(* IEC 61131-3 sources: Mizera_Tube/Plc (part 4) *)

(* ---- OUnSu.plc ---- *)
#funcdec "assi.plc"
#funcdec "DynMng.plc"
#funcdec "FBAux.plc"
#funcdec "SupForce.plc"
#funcdec "OSuppFB.plc"

VAR
#include "iof.inc"
#include "usrIof.inc"
#include "cnc.inc"

* Axis support management
* CN7 -> YUVW ( 85,86,87,88 ) Horizontal Supports
* CN8 -> YUVW ( 72,73,74,75 ) Correspoding Vertical Supports

SUP85:        HOR_SUPPORT;
SUP86:        HOR_SUPPORT;
SUP87:        HOR_SUPPORT;
SUP88:        HOR_SUPPORT;

F_TRIG_RES_FOLL:   F_TRIG;
END_VAR

VAR_IN_OUT
#include "usrIol.inc"
#include "mem.inc"
END_VAR

#include "Iol.inc"
#include "usrMem.inc"

FUNCTION HORIZ_SUPP

PATH %cn7

*******************************************************
*     HORIZONTAL FOLLOWIING SUPPORTS MANAGEMENT       *
*******************************************************
CAL  F_TRIG_RES_FOLL (CLK:=PRGRUN_CN0)
LD   F_TRIG_RES_FOLL.Q
OR   Pul_Reset
R    EnWriteBlendSwitch_Hor
R    CmdBlendSwitch_Hor

LDN  PRGRUN_CN0
JMPCN RSTBLEND
     LD   %PLCFLAGS.0
     ST   EnWriteBlendSwitch_Hor
     ST   CmdBlendSwitch_Hor
	 ST   iso_VshapeSecFollow
     ST   Iso_G520HorUnload_Ax85
     ST   Iso_G520HorUnload_Ax86
     ST   Iso_G520HorUnload_Ax87
     ST   Iso_G520HorUnload_Ax88
RSTBLEND:

LD   Reset
OR   EMER_GEN
ST   SUP85.xReset
ST   SUP86.xReset
ST   SUP87.xReset
ST   SUP88.xReset

LD   ISO_SupHor_Init
ST   SUP85.xHoldExem
ST   SUP86.xHoldExem
ST   SUP87.xHoldExem
ST   SUP88.xHoldExem

LDN  OptJogNoAutoHorPrk
ST   SUP85.xEnJogPrk
ST   SUP86.xEnJogPrk
ST   SUP87.xEnJogPrk
ST   SUP88.xEnJogPrk

LD   EnWriteBlendSwitch_Hor
AND  CmdBlendSwitch_Hor
ST   SUP85.xBlendSwitchEn
ST   SUP86.xBlendSwitchEn
ST   SUP87.xBlendSwitchEn
ST   SUP88.xBlendSwitchEn

LD   OptEnabAutoPark
ST   SUP85.xEnabAutoDwn
ST   SUP86.xEnabAutoDwn
ST   SUP87.xEnabAutoDwn
ST   SUP88.xEnabAutoDwn
ST   SUP85.xEnabAutoUp
ST   SUP86.xEnabAutoUp
ST   SUP87.xEnabAutoUp
ST   SUP88.xEnabAutoUp

LD   %ax85.pa22
ST   SUP85.xParkingPos
ST   SUP86.xParkingPos
ST   SUP87.xParkingPos
ST   SUP88.xParkingPos

LD   UnSupHorSafeZone
ST   SUP85.xColiQta
ST   SUP86.xColiQta
ST   SUP87.xColiQta
ST   SUP88.xColiQta

* For Vshape unloading only

LD   iso_VshapeSecFollow
ST   SUP85.xEnSecFollow
ST   SUP86.xEnSecFollow
ST   SUP87.xEnSecFollow
ST   SUP88.xEnSecFollow

LD   VShapeHorOffest
ST   SUP85.xAddFollPos
ST   SUP86.xAddFollPos
ST   SUP87.xAddFollPos
ST   SUP88.xAddFollPos

* [lv, lat, ulv, uhor]=[0,1,2,3]
LD   3
ST   SUP85.xBlendId
ST   SUP86.xBlendId
ST   SUP87.xBlendId
ST   SUP88.xBlendId

LD   iso_G520_Running
ST   SUP85.xEnBldFeed
ST   SUP86.xEnBldFeed
ST   SUP87.xEnBldFeed
ST   SUP88.xEnBldFeed

LD   100
ST   SUP85.xBldFeed
ST   SUP86.xBldFeed
ST   SUP87.xBldFeed
ST   SUP88.xBldFeed

* Horizontal Unloading Speed Control
LD   HorUnloadingFeed
GT   0
AND(
LD   HorUnloadingFeed
LE   100
)
JMPCN _HORFEEDCONTROL
     LD   HorUnloadingFeed
     ST   SUP85.xBldFeed
     ST   SUP86.xBldFeed
     ST   SUP87.xBldFeed
     ST   SUP88.xBldFeed
_HORFEEDCONTROL:

*******************************************************
* Support 1
*******************************************************
LD   %cn7.cc1.2
JMPCN no_support_85

PATH %ax85

LD   Z2Supp_72InParkPos
ST   SUP85.xVerParked

LD   Hold_U_Z2Supp
ST   SUP85.xHoldSuperviAxis

LD   HoldZ2Supp
ST   SUP85.xHoldSuppAxis

LD   SUP72_xParkCmd
ANDN iso_G520_Running
OR   Iso_G520HorUnload_Ax85
AND  %cn0.rc8.0
ST   SUP85.xParkCmd

CAL  SUP85

LD   SUP85.yReqGrant
ANDN ch7_in_ref
ST   usrReqGrantSupHorAx85

LD   SUP85.yHoldMovSupp
ANDN ch7_in_ref
ST   HoldSuppUn_HorAx85

LD   SUP85.yHoldMovSuperv
ANDN ch7_in_ref
ST   Hold_U_SupUnHorAx85

LD   SUP85.yVerForceDwn
ANDN ch7_in_ref
ST   Hor_Ax72_yVerForceDwn

no_support_85:

*******************************************************
* Support 2
*******************************************************
LD   %cn7.cc1.3
JMPCN no_support_86

PATH  %ax86

LD   Z3Supp_73InParkPos
ST   SUP86.xVerParked

LD   Hold_U_Z3Supp
ST   SUP86.xHoldSuperviAxis

LD   HoldZ3Supp
ST   SUP86.xHoldSuppAxis

LD   SUP73_xParkCmd
ANDN iso_G520_Running
OR   Iso_G520HorUnload_Ax86
AND  %cn0.rc8.0
ST   SUP86.xParkCmd

CAL  SUP86

LD   SUP86.yReqGrant
ANDN ch7_in_ref
ST   usrReqGrantSupHorAx86

LD   SUP86.yHoldMovSupp
ANDN ch7_in_ref
ST   HoldSuppUn_HorAx86

LD   SUP86.yHoldMovSuperv
ANDN ch7_in_ref
ST   Hold_U_SupUnHorAx86

LD   SUP86.yVerForceDwn
ANDN ch7_in_ref
ST   Hor_Ax73_yVerForceDwn

no_support_86:

*******************************************************
* Support 3
*******************************************************
LD   %cn7.cc1.4
JMPCN no_support_87

PATH  %ax87

LD   Z4Supp_74InParkPos
ST   SUP87.xVerParked

LD   Hold_U_Z4Supp
ST   SUP87.xHoldSuperviAxis

LD   HoldZ4Supp
ST   SUP87.xHoldSuppAxis

LD   SUP74_xParkCmd
ANDN iso_G520_Running
OR   Iso_G520HorUnload_Ax87
AND  %cn0.rc8.0
ST   SUP87.xParkCmd

CAL  SUP87

LD   SUP87.yReqGrant
ANDN ch7_in_ref
ST   usrReqGrantSupHorAx87

LD   SUP87.yHoldMovSupp
ANDN ch7_in_ref
ST   HoldSuppUn_HorAx87

LD   SUP87.yHoldMovSuperv
ANDN ch7_in_ref
ST   Hold_U_SupUnHorAx87

LD   SUP87.yVerForceDwn
ANDN ch7_in_ref
ST   Hor_Ax74_yVerForceDwn

no_support_87:

*******************************************************
* Support 4
*******************************************************
LD   %cn7.cc1.5
JMPCN no_support_88

PATH  %ax88

LD   Z5Supp_75InParkPos
ST   SUP88.xVerParked

LD   Hold_U_Z5Supp
ST   SUP88.xHoldSuperviAxis

LD   HoldZ5Supp
ST   SUP88.xHoldSuppAxis

LD   SUP75_xParkCmd
ANDN iso_G520_Running
OR   Iso_G520HorUnload_Ax88
AND  %cn0.rc8.0
ST   SUP88.xParkCmd

CAL  SUP88

LD   SUP88.yReqGrant
ANDN ch7_in_ref
ST   usrReqGrantSupHorAx88

LD   SUP88.yHoldMovSupp
ANDN ch7_in_ref
ST   HoldSuppUn_HorAx88

LD   SUP88.yHoldMovSuperv
ANDN ch7_in_ref
ST   Hold_U_SupUnHorAx88

LD   SUP88.yVerForceDwn
ANDN ch7_in_ref
ST   Hor_Ax75_yVerForceDwn

no_support_88:

END_FUNCTION

(* ---- pageplc.plc ---- *)
#include "iol.inc"

VAR
appoggio:        BOOL;
TP_Tab_Note:     TP;
END_VAR

*/ pop out page to select mode after reset */

FUNCTION PAGE_PLC

LD     HMI_PagePop
ANDN   %PLCFLAGS.8
ANDN(
    LD     %Uipl.Page
    EQ     171501
)
JMPCN  POP_WIND_STATE
    LD     171501
    ST     %PlcPage

    LD     1
    S      %ChangePlcPageFlags.3

    LD     1400
    ST     %WidthUiplDlg

    LD     400
    ST     %HeightUiplDlg

    LD     1
    ST     %ChangePlcPage
JMPC   COM_WIND_STATE
POP_WIND_STATE:
    LD     0
    ST     %ChangePlcPage
COM_WIND_STATE:

LD HMI_Ret2Loader
ANDN(
    LD     %Uipl.Page
    EQ     171502           ** Ret2Load.str
)
JMPCN  Skip_Ret2Load
    LD     171502
    ST     %PlcPage

    LD     1
    S      %ChangePlcPageFlags.3

    LD     1400
    ST     %WidthUiplDlg

    LD     400
    ST     %HeightUiplDlg

    LD     1
    ST     %ChangePlcPage
JMPC   COM_WIND_STATE2
Skip_Ret2Load:
    LD     0
    ST     %ChangePlcPage
COM_WIND_STATE2:

LDN    %cn0.rc8.0
JMPCN  PGMNORUNNING
    LD     %PLCFLAGS.0
    ST     Gui_btn_NoGear
    ST     Gui_btn_Gear
    ST     HMI_PagePop
    ST     HMI_Ret2Loader
PGMNORUNNING:

LD     %Uipl.Page
EQ     171501
JMPCN  CLRPAGEREQ
    LD     %PLCFLAGS.0
    ST     HMI_PagePop
CLRPAGEREQ:

LD     %Uipl.Page
EQ     171502
JMPCN  CLRPAGEREQ2
    LD     %PLCFLAGS.0
    ST     HMI_Ret2Loader
CLRPAGEREQ2:

END_FUNCTION

(* ---- Pneumat.plc ---- *)
*******************************************************************************
*   PNEUMAT.PLC
*   ESAutomotion
*   LASER machine
*******************************************************************************
VAR
#include "Cnc.inc"

appoggio:                       BOOL;       * Appoggio
TON_NOARIA:                     TON;        * Manca aria compressa
Strobe_Funz_M493:               BOOL;
Strobe_Funz_M494:               BOOL;
Memo_Aria_ass_taglio_da_Funz_M: BOOL;       * Memoria Aria assistenza al taglio da Funzione M
Aria_ass_taglio_in_Piercing:    BOOL;       * Aria assistenza al taglio in Piercing
R_TRIG493:                      R_TRIG;     * Fronte di salita M493 Attivazione Aria assistenza al taglio
R_TRIG494:                      R_TRIG;     * Fronte di salita M494 Disattivazione Aria assistenza al taglio
Test_Aria_ass_taglio_da_GUI     AT  %LsGui18.1;     *Test Aria assistenza al taglio da GUI
Test_Aria_ugello_da_GUI         AT  %LsGui18.2;     * Test Aria ugello da GUI
END_VAR

#include "Iol.inc"

VAR_IN_OUT
#include "mem.inc"
END_VAR

*******************************************************************************
*   Gestione Impianto Pneumatico
*******************************************************************************
FUNCTION Pneumatico

*******************************************************************************
* Allarme: bassa pressione aria impianto
*******************************************************************************
LDN  I_I_PRESSIONE_ARIA_IMPIANTO   ** Pressione aria Impianto OK
ST   appoggio                      ** Appoggio

CAL  TON_NOARIA(IN=appoggio, PT=1000) ** Manca aria compressa

LD   TON_NOARIA.Q
S    %PLCerr6.1

LD   RESET_ALLARMI                 ** M100.4  Cancellazione allarmi attiva
R    %PLCerr6.1                            ** PLC Err 193 Bassa pressione aria impianto

*******************************************************************************
* Allarme: bassa pressione aria banco
*******************************************************************************
LDN  I_I_PRESSIONE_ARIA_BANCO      ** Pressione aria Banco OK
S    %PLCerr6.2                            ** PLC Err 194 Bassa pressione aria banco

LD   RESET_ALLARMI                 ** M100.4  Cancellazione allarmi attiva
R    %PLCerr6.2                            ** PLC Err 194 Bassa pressione aria banco

*******************************************************************************
* Aria ugello : M498\M497 : Dis\Attivazione (IN Gas.plc)
*******************************************************************************
LD   GAS_prun                      ** M107.1 Cutting gas active from part program
ANDN %PlcOp0.2                     ** DryRun
ANDN PRGSTOP_CN0                   ** (cn0.rc8.1)  Programma interrotto CN0
OR   Test_Aria_ugello_da_GUI       ** Test Aria ugello da GUI
ST   O_O_EV_ARIA_UGELLO            ** Elettrovalvola aria ugello

*******************************************************************************
* Aria assistenza al taglio : M494\M493 : Dis\Attivazione
*******************************************************************************
LD   %cn0.rc9                               ** Channel 0 M-Functions register
EQ   493
AND  %cn0.rc8.4                             ** Channel 0 M-Functions Strobe
ST   Strobe_Funz_M493

CAL R_TRIG493(CLK=Strobe_Funz_M493) ** Fronte di salita M493 Attivazione Aria assistenza al taglio

LD   %cn0.rc9                               ** Channel 0 M-Functions register
EQ   494
AND  %cn0.rc8.4                             ** Channel 0 M-Functions Strobe
ST   Strobe_Funz_M494

CAL  R_TRIG494(CLK=Strobe_Funz_M494) ** Fronte di salita M494 Disattivazione Aria assistenza al taglio

LD   R_TRIG493.Q
S    Memo_Aria_ass_taglio_da_Funz_M ** Memoria Aria assistenza al taglio da Funzione M
LD   R_TRIG494.Q
ORN  MACCHINA_OK                   ** M100.1  Macchina OK
OR   RESET_MACCHINA                ** M100.2  Reset macchina
R    Memo_Aria_ass_taglio_da_Funz_M ** Memoria Aria assistenza al taglio da Funzione M

LD   %TabLsr0.L_UserInt1
EQ   0
ST   Aria_ass_taglio_in_Piercing   ** Aria assistenza al taglio in Piercing

LD   Memo_Aria_ass_taglio_da_Funz_M ** Memoria Aria assistenza al taglio da Funzione M
OR   Aria_ass_taglio_in_Piercing   ** Aria assistenza al taglio in Piercing
AND(
LD   PRGRUN_CN0                    ** M0.0 cn0.rc8.0  Programma in corso
ANDN %PlcOp0.2                     ** DryRun
ANDN PRGSTOP_CN0                   ** (cn0.rc8.1)  Programma interrotto CN0
ANDN ExeAuxMode                    ** (gPlc0.29)Esecuzione ausiliaria 1000.PGM
)
OR   Test_Aria_ass_taglio_da_GUI   ** Test Aria assistenza al taglio da GUI
ST   O_O_EV_ASSISTENZA_TAGLIO      ** Elettrovalvola assistenza taglio

*******************************************************************************
*Segnalazioni per Aggiornamento pagina video
*******************************************************************************
LD   O_O_EV_ARIA_UGELLO            ** Elettrovalvola aria ugello
ST   GasYV23LED                    ** (LsPlc11.12) LED nozzle air

LD   O_O_EV_ASSISTENZA_TAGLIO      ** Elettrovalvola assistenza taglio
ST   GasYV24LED                    ** (LsPlc11.13) LED cut air assistance

END_FUNCTION

(* ---- remcon.plc ---- *)
#include "Iol.inc"

VAR
#include "Cnc.inc"
#include "RemContr.inc"
END_VAR

VAR
DryrunSig                  AT %PlcOp0.2 ; ** DryRun
HoldingZ                   AT %ax29.ra0.1;                  * %ax29.ra0.1 holding Z axis
HoldingX                   AT %ax27.ra0.1;                  * %ax27.ra0.1 holding X axis
HoldingY                   AT %ax28.ra0.1;                  * %ax29.ra0.1 holding Y axis
END_VAR

FUNCTION REMOTE_DISPLAY
******************************************************************************
* THE AXIS DISPLAY
******************************************************************************
LD   %ax30.ra4                   *U position Yang
DIV  10
ST   X_AXIS_POSITION

LD   %ax28.ra4
DIV  10
ST   Y_AXIS_POSITION

LD   %ax29.ra4
DIV  10
ST   Z_AXIS_POSITION

LD      HoldingZ                   ** %ax29.ra0.1 holding Z axis
JMPCN   Z_HOLDING
LD      4
ST      LineZaxis                  ** XhcApp.Xhc_LineIdx3 Feedrate and mode
JMP     END_AZ
Z_HOLDING:
LD      1
ST      LineZaxis                  ** XhcApp.Xhc_LineIdx3 Feedrate and mode
END_AZ:

LD      HoldingX                   ** %ax27.ra0.1 holding X axis
JMPCN   X_HOLDING
LD      5
ST      LineXaxis                  ** XhcApp.Xhc_LineIdx1 X axis quote
JMP     END_AX
X_HOLDING:
LD      2
ST      LineXaxis                  ** XhcApp.Xhc_LineIdx1 X axis quote
END_AX:

LD      HoldingY                   ** %ax29.ra0.1 holding Y axis
JMPCN   Y_HOLDING
LD      6
ST      LineYaxis                  ** XhcApp.Xhc_LineIdx2 Y axis quote
JMP     END_AY
Y_HOLDING:
LD      3
ST      LineYaxis                  ** XhcApp.Xhc_LineIdx2 Y axis quote
END_AY:

******************************************************************************
* THE FEEDRATE DISPLAY
******************************************************************************
LD       DryrunSig                 ** %PlcOp0.2 Dry signal
AND      BCI_TAR                   * rc0.8  Selettore modi operativi su REF (taratura)
JMPCN    DRY_REF
LD       12
ST       LineFeed                  ** XhcApp.Xhc_LineIdx0 Z axis quote
JMP      END_CONDITION
DRY_REF:

LDN      DryrunSig                 ** %PlcOp0.2 Dry signal
AND      BCI_TAR                   * rc0.8  Selettore modi operativi su REF (taratura)
JMPCN    NOTDRY_REF
LD       7
ST       LineFeed                  ** XhcApp.Xhc_LineIdx0 Z axis quote
JMP      END_CONDITION
NOTDRY_REF:

LD       DryrunSig                 ** %PlcOp0.2 Dry signal
AND      BCI_MAN                   * rc0.9  Selettore modi operativi su JOG (manuale)
JMPCN    DRY_JOG
LD       13
ST       LineFeed                  ** XhcApp.Xhc_LineIdx0 Z axis quote
JMP      END_CONDITION
DRY_JOG:

LDN      DryrunSig                 ** %PlcOp0.2 Dry signal
AND      BCI_MAN                   * rc0.9  Selettore modi operativi su JOG (manuale)
JMPCN    NOTDRY_JOG
LD       8
ST       LineFeed                  ** XhcApp.Xhc_LineIdx0 Z axis quote
JMP      END_CONDITION
NOTDRY_JOG:

LD       DryrunSig                 ** %PlcOp0.2 Dry signal
AND      BCI_INC                   * rc0.10  Selettore modi operativi su INC (inc.fissi)
JMPCN    DRY_INC
LD       14
ST       LineFeed                  ** XhcApp.Xhc_LineIdx0 Z axis quote
JMP      END_CONDITION
DRY_INC:

LDN      DryrunSig                 ** %PlcOp0.2 Dry signal
AND      BCI_INC                   * rc0.10  Selettore modi operativi su INC (inc.fissi)
JMPCN    NOTDRY_INC
LD       9
ST       LineFeed                  ** XhcApp.Xhc_LineIdx0 Z axis quote
JMP      END_CONDITION
NOTDRY_INC:

LD       DryrunSig                 ** %PlcOp0.2 Dry signal
AND      BCI_MDI                   * rc0.11  Selettore modi operativi su MDI (semiautom)
JMPCN    DRY_MDI
LD       15
ST       LineFeed                  ** XhcApp.Xhc_LineIdx0 Z axis quote
JMP      END_CONDITION
DRY_MDI:

LDN      DryrunSig                 ** %PlcOp0.2 Dry signal
AND      BCI_MDI                   * rc0.11  Selettore modi operativi su MDI (semiautom)
JMPCN    NOTDRY_MDI
LD       10
ST       LineFeed                  ** XhcApp.Xhc_LineIdx0 Z axis quote
JMP      END_CONDITION
NOTDRY_MDI:

LD       DryrunSig                 ** %PlcOp0.2 Dry signal
AND      BCI_AUT                   * rc0.12  Selettore modi operativi su AUT (automatic)
JMPCN    DRY_AUT
LD       16
ST       LineFeed                  ** XhcApp.Xhc_LineIdx0 Z axis quote
JMP      END_CONDITION
DRY_AUT:

LDN      DryrunSig                 ** %PlcOp0.2 Dry signal
AND      BCI_AUT                   * rc0.12  Selettore modi operativi su AUT (automatic)
JMPCN    NOTDRY_AUT
LD       11
ST       LineFeed                  ** XhcApp.Xhc_LineIdx0 Z axis quote

NOTDRY_AUT:

END_CONDITION:

END_FUNCTION

(* ---- RemContr.plc ---- *)
*******************************************************************************
*   RemContR.plc
*   ESAutomotion
*   LASER machine
*   Remote Controller Manag
*******************************************************************************
#funcdec "FLP.plc"

VAR
#include "RemContr.inc"
END_VAR

#include "Iol.inc"

VAR_IN_OUT
#include "mem.inc"
END_VAR

FUNCTION   REMOTE_CONTROLLER

(* ---- resmach.plc ---- *)
*******************************************************************************
*   RESMACH.PLC
*   ESAutomotion
*   LASER machine
*******************************************************************************
*
* Reset function
* There is update:
* To Reset Axes with TON maybe OK, but CN Reset should check real feedback
* Res_Ch3 is also used to xReset CN4 on this machine
*
* Reset must be:
* 1) Disable gearing to unlock real axes from virtual axes,
* 2) Reset channel 3 4
* 3) Reset channel 0 2 5
*******************************************************************************
#funcdec "assi.plc"
#funcdec "cnc.plc"

VAR
#include "assi.inc"
#include "cnc.inc"

END_VAR

VAR_IN_OUT
#include "mem.inc"
END_VAR

#include "iol.inc"

VAR
RTRIG_RESET:        R_TRIG;
TON_RES_AXES:       TON;
TON_RESCH3:         TON;
TON_RESCH0:         TON;
ResetCh0Ok:         BOOL;
ResetCh3Ok:         BOOL;
check_ch3:          BOOL;
END_VAR

*******************************************************************************
FUNCTION  MACHINE_RESET

LDN  %cn0.rc8.0
ANDN %cn0.rc8.1
ST   ResetCh0Ok

LDN  %cn3.rc8.0
ANDN %cn3.rc8.1
ST   ResetCh3Ok

CAL  RTRIG_RESET(CLK:=ResetMach)          * Reset pushbutton

LD   RTRIG_RESET.Q
S    Res_Axes

CAL  TON_RES_AXES(IN:=Res_Axes,PT:=200)
LD   TON_RES_AXES.Q
***OR(
***LD   ResetCh0Ok
***ANDN ResetCh3Ok
***)
R    Res_Axes
R    check_ch3
S    Res_Ch3

* In Main, not to allow START with any Res_

CAL  TON_RESCH3(IN:=Res_Ch3,PT:=200)
LD   TON_RESCH3.Q
S    check_ch3
R    Res_Ch3

LD   check_ch3
AND  %cn3.rc8.21
R    check_ch3
S    Res_Ch0

CAL  TON_RESCH0(IN:=Res_Ch0,PT:=200)
LD   TON_RESCH0.Q
R    Res_Ch0

END_FUNCTION

(* ---- SupLdCy.plc ---- *)
#funcdec "FBSuppor.plc"
#funcdec "assi.plc"
#funcdec "DynMng.plc"
#funcdec "FBAux.plc"
#funcdec "SupForce.plc"
#funcdec "suppFB.plc"

#include "Iol.inc"
#include "usrMem.inc"

VAR
#include "iof.inc"
#include "usrIof.inc"
#include "cnc.inc"

SUPPORT_1:     TUBE_SUPPORT;
SUPPORT_2:     TUBE_SUPPORT;
SUPPORT_3:     TUBE_SUPPORT;
SUPPORT_4:     TUBE_SUPPORT;
SUPPORT_5:     TUBE_SUPPORT;
SUPPORT_6:     TUBE_SUPPORT;
SUPPORT_7:     TUBE_SUPPORT;
END_VAR

VAR_IN_OUT
#include "usrIol.inc"
#include "mem.inc"
END_VAR

FUNCTION LOAD_CYLINDER_SUPPORTS

*******************************************************
*           CYLINDER SUPPORTS MANAGEMENT              *
*******************************************************
LD   SUPPORTS_JogPlus
ST   SUPPORTS_JogPlusLed

LD   SUPPORTS_JogMinus
ST   SUPPORTS_JogMinusLed

LD   ALWAYS_ONE
ST   SUPPORT_1.xUaxDir
ST   SUPPORT_2.xUaxDir
ST   SUPPORT_3.xUaxDir
ST   SUPPORT_4.xUaxDir

LD   PosUMis
ST   SUPPORT_1.xPosU
ST   SUPPORT_2.xPosU
ST   SUPPORT_3.xPosU
ST   SUPPORT_4.xPosU

LD   ThreshLoadingSupDown
ST   SUPPORT_1.xSuperviseOft
ST   SUPPORT_2.xSuperviseOft
ST   SUPPORT_3.xSuperviseOft
ST   SUPPORT_4.xSuperviseOft

LDN  I_I_EMERGENZA                ** Machine OK (no EMERG.)
ST   SUPPORT_1.xEmerg
ST   SUPPORT_2.xEmerg
ST   SUPPORT_3.xEmerg
ST   SUPPORT_4.xEmerg

LD   ch0_in_aut                   ** channel 0 in aut
ST   SUPPORT_1.xAuto
ST   SUPPORT_2.xAuto
ST   SUPPORT_3.xAuto
ST   SUPPORT_4.xAuto

LD   I_I_PRESSIONE_ARIA_IMPIANTO
ST   SUPPORT_1.xAirPressure
ST   SUPPORT_2.xAirPressure
ST   SUPPORT_3.xAirPressure
ST   SUPPORT_4.xAirPressure

LD   Reset                        ** Reset Command
OR   Start_Ch0                    ** Start Request to Ch0
ST   SUPPORT_1.xReset
ST   SUPPORT_2.xReset
ST   SUPPORT_3.xReset
ST   SUPPORT_4.xReset

LD   TimeOutPistonDown
ST   SUPPORT_1.xTimeOut
ST   SUPPORT_2.xTimeOut
ST   SUPPORT_3.xTimeOut
ST   SUPPORT_4.xTimeOut

*******************************************************
*                      SUPPORT 1                      *
*******************************************************
LD   I_I_Support_1_Dwn            ** M50.7 Support 1 Down Sensor
ST   SUPPORT_1.xSensorDwn

LD   I_I_Support_1_Up
ST   SUPPORT_1.xSensorOpen

LD   SUPPORTS_S1_Selected
AND  SUPPORTS_JogPlus
ST   SUPPORT_1.xManualUp

LD   SUPPORTS_S1_Selected
AND  SUPPORTS_JogMinus
ST   SUPPORT_1.xManualDwn

LD   Fun_M724_Ch0                 ** Auto Up command for supports
OR   Fun_M733_Ch0
ANDN yActivatedCyCom_51
ST   SUPPORT_1.xAutoUp

LD   Fun_M725_Ch0                 ** Auto Up command for supports
OR   yActivatedCyCom_51
ST   SUPPORT_1.xAutoDwn

LD   SUPPORT_1_AutoEnable
ST   SUPPORT_1.xEnable

LD   SUPPORT_1_Quota
ST   SUPPORT_1.xLimitQuota

CAL  SUPPORT_1

LD   SUPPORT_1.yEvUp
ST   O_O_Ev_Support1_Up

LD   SUPPORT_1.yEvDwn
ST   O_O_Ev_Support1_Dwn

LD   SUPPORT_1.yAlarmDwn
ST   SUPPORT_1_AlarmDwn
ST   %PLCerr21.0

*******************************************************
*                      SUPPORT 2                      *
*******************************************************
LD   I_I_Support_2_Dwn             ** M50.8 Support 2 Down Sensor
ST   SUPPORT_2.xSensorDwn

LD   I_I_Support_2_Up              ** PLCFLAGS.1  Flag sempre stato on
ST   SUPPORT_2.xSensorOpen

LD   SUPPORTS_S2_Selected
AND  SUPPORTS_JogPlus
ST   SUPPORT_2.xManualUp

LD   SUPPORTS_S2_Selected
AND  SUPPORTS_JogMinus
ST   SUPPORT_2.xManualDwn

LD   Fun_M724_Ch0                  ** Auto Up command for supports
OR   Fun_M734_Ch0
ANDN yActivatedCyCom_52
ST   SUPPORT_2.xAutoUp

LD   Fun_M725_Ch0                  ** Auto Up command for supports
OR   yActivatedCyCom_52
ST   SUPPORT_2.xAutoDwn

LD   SUPPORT_2_AutoEnable
ST   SUPPORT_2.xEnable

LD   SUPPORT_2_Quota
ST   SUPPORT_2.xLimitQuota

CAL  SUPPORT_2

LD   SUPPORT_2.yAlarmDwn
ST   SUPPORT_2_AlarmDwn
ST   %PLCerr21.1

LD   SUPPORT_2.yEvUp
ST   O_O_Ev_Support2_Up

LD   SUPPORT_2.yEvDwn
ST   O_O_Ev_Support2_Dwn

*******************************************************
*                      SUPPORT 3                      *
*******************************************************
LD   I_I_Support_3_Dwn             ** M50.9 Support 3 Down Sensor
ST   SUPPORT_3.xSensorDwn

LD   I_I_Support_3_Up
ST   SUPPORT_3.xSensorOpen

LD   SUPPORTS_S3_Selected
AND  SUPPORTS_JogPlus
ST   SUPPORT_3.xManualUp

LD   SUPPORTS_S3_Selected
AND  SUPPORTS_JogMinus
ST   SUPPORT_3.xManualDwn

LD   Fun_M724_Ch0                  ** Auto Up command for supports
OR   Fun_M735_Ch0
ANDN yActivatedCyCom_53
ST   SUPPORT_3.xAutoUp

LD   Fun_M725_Ch0                  ** Auto Up command for supports
OR   yActivatedCyCom_53
ST   SUPPORT_3.xAutoDwn

LD   SUPPORT_3_AutoEnable
ST   SUPPORT_3.xEnable

LD   SUPPORT_3_Quota
ST   SUPPORT_3.xLimitQuota

CAL  SUPPORT_3

LD   SUPPORT_3.yAlarmDwn
ST   SUPPORT_3_AlarmDwn
ST   %PLCerr21.2

LD   SUPPORT_3.yEvUp
ST   O_O_Ev_Support3_Up

LD   SUPPORT_3.yEvDwn
ST   O_O_Ev_Support3_Dwn

*******************************************************
*                      SUPPORT 4                      *
*******************************************************
LD   I_I_Support_4_Dwn             ** M50.10 Support 4 Down Sensor
ST   SUPPORT_4.xSensorDwn

LD   I_I_Support_4_Up              ** PLCFLAGS.1  Flag sempre stato on
ST   SUPPORT_4.xSensorOpen

LD   SUPPORTS_S4_Selected
AND  SUPPORTS_JogPlus
ST   SUPPORT_4.xManualUp

LD   SUPPORTS_S4_Selected
AND  SUPPORTS_JogMinus
ST   SUPPORT_4.xManualDwn

LD   Fun_M724_Ch0                  ** Auto Up command for supports
OR   Fun_M736_Ch0
ANDN yActivatedCyCom_54
ST   SUPPORT_4.xAutoUp

LD   Fun_M725_Ch0                  ** Auto Up command for supports
OR   yActivatedCyCom_54
ST   SUPPORT_4.xAutoDwn

LD   SUPPORT_4_AutoEnable
ST   SUPPORT_4.xEnable

LD   SUPPORT_4_Quota
ST   SUPPORT_4.xLimitQuota

CAL  SUPPORT_4

LD   SUPPORT_4.yAlarmDwn
ST   SUPPORT_4_AlarmDwn
ST   %PLCerr21.3

LD   SUPPORT_4.yEvUp
ST   O_O_Ev_Support4_Up

LD   SUPPORT_4.yEvDwn
ST   O_O_Ev_Support4_Dwn

*******************************************************
*                    HOLD CONDITION                   *
*******************************************************
LD   %PLCerr21.0
OR   %PLCerr21.1
OR   %PLCerr21.2
OR   %PLCerr21.3
OR   %PLCerr21.4
OR   %PLCerr21.5
OR   %PLCerr21.6
OR   SUPPORT_1.yHoldMovSuperv
OR   SUPPORT_2.yHoldMovSuperv
OR   SUPPORT_3.yHoldMovSuperv
OR   SUPPORT_4.yHoldMovSuperv
ST   M_HoldAx_U

LD   I_I_Support_1_Dwn
AND  I_I_Support_2_Dwn
AND  I_I_Support_3_Dwn
AND  I_I_Support_4_Dwn
*AND  I_I_Support_5_Dwn
*AND  I_I_Support_6_Dwn
*AND  I_I_Support_7_Dwn
ST   All_Sup_DWN

END_FUNCTION

(* ---- SuUnCy.plc ---- *)
*******************************************************
*  Motor-cylinder Composite Support (Cylinder Part)   *
*  Supports Up/Dwn Conditions Based On Motor Part     *
*******************************************************
#funcdec "FBSuppor.plc"
#funcdec "assi.plc"
#funcdec "DynMng.plc"
#funcdec "FBAux.plc"
#funcdec "SupForce.plc"
#funcdec "suppFB.plc"

#include "Iol.inc"
#include "usrMem.inc"

VAR
#include "iof.inc"
#include "usrIof.inc"
#include "cnc.inc"

SUPPORT_71:     TUBE_SUPPORT;
SUPPORT_72:     TUBE_SUPPORT;
SUPPORT_73:     TUBE_SUPPORT;
SUPPORT_74:     TUBE_SUPPORT;
SUPPORT_75:     TUBE_SUPPORT;
END_VAR

VAR_IN_OUT
#include "usrIol.inc"
#include "mem.inc"
END_VAR

FUNCTION UN_CYLINDER_SUPPORTS
*******************************************************
*    UNLOAD CYLINDER SUPPORTS MANAGEMENT              *
*******************************************************
LD   UNSUPPORTS_JogPlus
ST   UNSUPPORTS_JogPlusLed

LD   UNSUPPORTS_JogMinus
ST   UNSUPPORTS_JogMinusLed

LD   SupervisePos_X1
ST   SUPPORT_71.xPosU
ST   SUPPORT_72.xPosU
ST   SUPPORT_73.xPosU
ST   SUPPORT_74.xPosU
ST   SUPPORT_75.xPosU

LDN  I_I_EMERGENZA
ST   SUPPORT_71.xEmerg
ST   SUPPORT_72.xEmerg
ST   SUPPORT_73.xEmerg
ST   SUPPORT_74.xEmerg
ST   SUPPORT_75.xEmerg

LD   ch0_in_aut
ST   SUPPORT_71.xAuto
ST   SUPPORT_72.xAuto
ST   SUPPORT_73.xAuto
ST   SUPPORT_74.xAuto
ST   SUPPORT_75.xAuto

LD   I_I_PRESSIONE_ARIA_IMPIANTO
ST   SUPPORT_71.xAirPressure
ST   SUPPORT_72.xAirPressure
ST   SUPPORT_73.xAirPressure
ST   SUPPORT_74.xAirPressure
ST   SUPPORT_75.xAirPressure

LD   Reset
OR   Start_Ch0
ST   SUPPORT_71.xReset
ST   SUPPORT_72.xReset
ST   SUPPORT_73.xReset
ST   SUPPORT_74.xReset
ST   SUPPORT_75.xReset

LD   TimeOutPistonDown
ST   SUPPORT_71.xTimeOut
ST   SUPPORT_72.xTimeOut
ST   SUPPORT_73.xTimeOut
ST   SUPPORT_74.xTimeOut
ST   SUPPORT_75.xTimeOut

*******************************************************
* Support On Ax71
*******************************************************
LD   I_I_SUPPORT_71_Dwn
ST   SUPPORT_71.xSensorDwn

LD   I_I_SUPPORT_71_Up
ST   SUPPORT_71.xSensorOpen

LD   SUPPORTS_S71_Selected
AND  UNSUPPORTS_JogPlus
ST   SUPPORT_71.xManualUp

LD   SUPPORTS_S71_Selected
AND  UNSUPPORTS_JogMinus
ST   SUPPORT_71.xManualDwn

LDN  Hold_U_Z1Supp
ANDN SUP71_xParkCmd
ANDN yActivatedCyCom_71
ST   SUPPORT_71.xAutoUp

LD   Hold_U_Z1Supp
OR   SUP71_xParkCmd
OR   yActivatedCyCom_71
ST   SUPPORT_71.xAutoDwn

LD   SUPPORT_71_AutoEnable
ST   SUPPORT_71.xEnable

LD   OffsetUnSuppDwn_71
ST   SUPPORT_71.xSuperviseOft

LD   U_Posit_Z1_Down
ST   SUPPORT_71.xLimitQuota

CAL  SUPPORT_71

LD   SUPPORT_71.yEvUp
ST   O_O_Ev_Support71_Up

LD   SUPPORT_71.yEvDwn
ST   O_O_Ev_Support71_Dwn

LD   SUPPORT_71.yAlarmDwn
ST   %PLCerr20.4

*******************************************************
* Support On Ax72
*******************************************************
LD   I_I_SUPPORT_72_Dwn
ST   SUPPORT_72.xSensorDwn

LD   I_I_SUPPORT_72_Up
ST   SUPPORT_72.xSensorOpen

LD   SUPPORTS_S72_Selected
AND  UNSUPPORTS_JogPlus
ST   SUPPORT_72.xManualUp

LD   SUPPORTS_S72_Selected
AND  UNSUPPORTS_JogMinus
ST   SUPPORT_72.xManualDwn

LDN  Hold_U_Z2Supp
ANDN SUP72_xParkCmd
ANDN yActivatedCyCom_72
ST   SUPPORT_72.xAutoUp

LD   Hold_U_Z2Supp
OR   SUP72_xParkCmd
OR   yActivatedCyCom_72
ST   SUPPORT_72.xAutoDwn

LD   SUPPORT_72_AutoEnable
ST   SUPPORT_72.xEnable

LD   OffsetUnSuppDwn_72
ST   SUPPORT_72.xSuperviseOft

LD   U_Posit_Z2_Down
ST   SUPPORT_72.xLimitQuota

CAL  SUPPORT_72

LD   SUPPORT_72.yEvUp
ST   O_O_Ev_Support72_Up

LD   SUPPORT_72.yEvDwn
ST   O_O_Ev_Support72_Dwn

LD   SUPPORT_72.yAlarmDwn
ST   %PLCerr20.5

*******************************************************
* Support On Ax73
*******************************************************
LD   I_I_SUPPORT_73_Dwn
ST   SUPPORT_73.xSensorDwn

LD   I_I_SUPPORT_73_Up
ST   SUPPORT_73.xSensorOpen

LD   SUPPORTS_S73_Selected
AND  UNSUPPORTS_JogPlus
ST   SUPPORT_73.xManualUp

LD   SUPPORTS_S73_Selected
AND  UNSUPPORTS_JogMinus
ST   SUPPORT_73.xManualDwn

LDN  Hold_U_Z3Supp
ANDN SUP73_xParkCmd
ANDN yActivatedCyCom_73
ST   SUPPORT_73.xAutoUp

LD   Hold_U_Z3Supp
OR   SUP73_xParkCmd
OR   yActivatedCyCom_73
ST   SUPPORT_73.xAutoDwn

LD   SUPPORT_73_AutoEnable
ST   SUPPORT_73.xEnable

LD   OffsetUnSuppDwn_73
ST   SUPPORT_73.xSuperviseOft

LD   U_Posit_Z3_Down
ST   SUPPORT_73.xLimitQuota

CAL  SUPPORT_73

LD   SUPPORT_73.yEvUp
ST   O_O_Ev_Support73_Up

LD   SUPPORT_73.yEvDwn
ST   O_O_Ev_Support73_Dwn

LD   SUPPORT_73.yAlarmDwn
ST   %PLCerr20.6

*******************************************************
* Support On Ax74
*******************************************************
LD   I_I_SUPPORT_74_Dwn
ST   SUPPORT_74.xSensorDwn

LD   I_I_SUPPORT_74_Up
ST   SUPPORT_74.xSensorOpen

LD   SUPPORTS_S74_Selected
AND  UNSUPPORTS_JogPlus
ST   SUPPORT_74.xManualUp

LD   SUPPORTS_S74_Selected
AND  UNSUPPORTS_JogMinus
ST   SUPPORT_74.xManualDwn

LDN  Hold_U_Z4Supp
ANDN SUP74_xParkCmd
ANDN yActivatedCyCom_74
ST   SUPPORT_74.xAutoUp

LD   Hold_U_Z4Supp
OR   SUP74_xParkCmd
OR   yActivatedCyCom_74
ST   SUPPORT_74.xAutoDwn

LD   SUPPORT_74_AutoEnable
ST   SUPPORT_74.xEnable

LD   OffsetUnSuppDwn_74
ST   SUPPORT_74.xSuperviseOft

LD   U_Posit_Z4_Down
ST   SUPPORT_74.xLimitQuota

CAL  SUPPORT_74

LD   SUPPORT_74.yEvUp
ST   O_O_Ev_Support74_Up

LD   SUPPORT_74.yEvDwn
ST   O_O_Ev_Support74_Dwn

LD   SUPPORT_74.yAlarmDwn
ST   %PLCerr20.7

*******************************************************
* Support On Ax75
*******************************************************
LD   I_I_SUPPORT_75_Dwn
ST   SUPPORT_75.xSensorDwn

LD   I_I_SUPPORT_75_Up
ST   SUPPORT_75.xSensorOpen

LD   SUPPORTS_S75_Selected
AND  UNSUPPORTS_JogPlus
ST   SUPPORT_75.xManualUp

LD   SUPPORTS_S75_Selected
AND  UNSUPPORTS_JogMinus
ST   SUPPORT_75.xManualDwn

LDN  Hold_U_Z5Supp
ANDN SUP75_xParkCmd
ANDN yActivatedCyCom_75
ST   SUPPORT_75.xAutoUp

LD   Hold_U_Z5Supp
OR   SUP75_xParkCmd
OR   yActivatedCyCom_75
ST   SUPPORT_75.xAutoDwn

LD   SUPPORT_75_AutoEnable
ST   SUPPORT_75.xEnable

LD   OffsetUnSuppDwn_75
ST   SUPPORT_75.xSuperviseOft

LD   U_Posit_Z5_Down
ST   SUPPORT_75.xLimitQuota

CAL  SUPPORT_75

LD   SUPPORT_75.yEvUp
ST   O_O_Ev_Support75_Up

LD   SUPPORT_75.yEvDwn
ST   O_O_Ev_Support75_Dwn

LD   SUPPORT_75.yAlarmDwn
ST   %PLCerr20.8

*******************************************************
*                    HOLD CONDITION                   *
*******************************************************
LD   %PLCerr20.4
OR   %PLCerr20.5
OR   %PLCerr20.6
OR   %PLCerr20.7
OR   %PLCerr20.8
OR   SUPPORT_71.yHoldMovSuperv
OR   SUPPORT_72.yHoldMovSuperv
OR   SUPPORT_73.yHoldMovSuperv
OR   SUPPORT_74.yHoldMovSuperv
OR   SUPPORT_75.yHoldMovSuperv
ST   M_HoldAx_V

END_FUNCTION

(* ---- UnFlaps.plc ---- *)
#funcdec "assi.plc"
#funcdec "suppFB.plc"
#funcdec "SPist.plc"
#funcdec "DynMng.plc"
#funcdec "FBAux.plc"
#funcdec "SupForce.plc"

#include "usrMem.inc"
#include "Iol.inc"

VAR
#include "iof.inc"
#include "usrIof.inc"
#include "cnc.inc"

FlapA71:              SINGLE_PISTON;
FlapA72:              SINGLE_PISTON;
FlapA73:              SINGLE_PISTON;
FlapA74:              SINGLE_PISTON;
FlapA75:              SINGLE_PISTON;
END_VAR

VAR_IN_OUT
#include "usrIol.inc"
#include "mem.inc"
END_VAR

FUNCTION UNLOAD_FLAPS

********************************************************************************
* UNLOAD FLAPS MANAGEMENT                                                      *
********************************************************************************
LD   PRGRUN_CN0                       ** M0.0 cn0.rc8.0  Programma in corso
ST   FlapA72.xAuto
ST   FlapA71.xAuto
ST   FlapA73.xAuto
ST   FlapA74.xAuto
ST   FlapA75.xAuto

LD   Pul_Reset                        ** (gPlc0.3)Reset pushbutton
OR   Pul_Start                        ** (gPlc0.1)Start pushbutton
ST   FlapA72.xReset
ST   FlapA71.xReset
ST   FlapA73.xReset
ST   FlapA74.xReset
ST   FlapA75.xReset

LD   I_I_PRESSIONE_ARIA_IMPIANTO      ** %USR_M0
ST   FlapA72.xAirPressure
ST   FlapA71.xAirPressure
ST   FlapA73.xAirPressure
ST   FlapA74.xAirPressure
ST   FlapA75.xAirPressure

LD   ALWAYS_ONE
ST   FlapA72.xPlusAtInit
ST   FlapA71.xPlusAtInit
ST   FlapA73.xPlusAtInit
ST   FlapA74.xPlusAtInit
ST   FlapA75.xPlusAtInit

LD   ALWAYS_ZERO                      ** PLCFLAGS.0  Flag sempre stato off
ST   FlapA72.xSingleEffect
ST   FlapA71.xSingleEffect
ST   FlapA73.xSingleEffect
ST   FlapA74.xSingleEffect
ST   FlapA75.xSingleEffect

LD   TimeOutPistonDown
ST   FlapA72.xTimeOut
ST   FlapA71.xTimeOut
ST   FlapA73.xTimeOut
ST   FlapA74.xTimeOut
ST   FlapA75.xTimeOut

LDN  I_I_EMERGENZA                    ** Machine OK (no EMERG.)
ST   FlapA72.xEmerg
ST   FlapA71.xEmerg
ST   FlapA73.xEmerg
ST   FlapA74.xEmerg
ST   FlapA75.xEmerg

********************************************************************************
* Ax72, Unloader Flap L2
********************************************************************************
LD   %ax71.ra4
GT  (
     LD  UnloadSupQta
     ADD 1000
)
OR   Fun_M993_Ch0
ST   ForceFlapUpZone

LD   Flap71JogHome
OR   AllFlapsHome
OR   ForceFlapUpZone
OR   ParkAllCmd
ST   FlapA71.xManualPlus

LD   Flap71JogIncline
OR   AllFlapsIncline
ANDN ForceFlapUpZone
ST   FlapA71.xManualMinus

LD   Fun_M829_Ch0                     ** Auto Up command for supports
OR   ForceFlapUpZone
OR   AllFlapsHome
ST   FlapA71.xAutoPlus

LD   Fun_M830_Ch0                     ** Auto DWN command for supports
OR   InclineFlapL1_ISO
ANDN ForceFlapUpZone
ST   FlapA71.xAutoMinus

LD   I_I_Flap_Home
ST   FlapA71.xSensorPlus

LD   I_I_Flap_Inclined                ** M57.1
ST   FlapA71.xSensorMinus

CAL  FlapA71

LD   FlapA71.yPistonPlus
OR   HoldFlapInclined
ST   O_O_Flap_Home

LD   FlapA71.yPistonMinus
ANDN HoldFlapInclined
ST   O_O_Flap_Incline

LD   FlapA71.yAlarm
AND  %cn8.cc1.1
ST   %PLCerr21.14

LD   ForceFlapUpZone
ST   ForceFlapUp_71

********************************************************************************
* Ax72, Unloader Flap L2
********************************************************************************
LD   %ax72.ra4
GT  (
     LD  UnloadSupQta
     ADD 1000
)
OR   Fun_M993_Ch0
ST   ForceFlapUpZone

LD   Flap72JogHome
OR   AllFlapsHome
OR   ForceFlapUpZone
OR   ParkAllCmd
ST   FlapA72.xManualPlus

LD   Flap72JogIncline
OR   AllFlapsIncline
ANDN ForceFlapUpZone
ST   FlapA72.xManualMinus

LD   Fun_M826_Ch0                     ** Auto Up command for supports
OR   ForceFlapUpZone
OR   AllFlapsHome
ST   FlapA72.xAutoPlus

LD   Fun_M827_Ch0                     ** Auto DWN command for supports
OR   InclineFlapL2_ISO
ANDN ForceFlapUpZone
ST   FlapA72.xAutoMinus

LD   I_I_FlapL2_Home
ST   FlapA72.xSensorPlus

LD   I_I_FlapL2_Inclined                ** M57.1
ST   FlapA72.xSensorMinus

CAL  FlapA72

LD   FlapA72.yPistonPlus
OR   HoldFlapInclined
ST   O_O_FlapL2_Home

LD   FlapA72.yPistonMinus
ANDN HoldFlapInclined
ST   O_O_FlapL2_Incline

LD   FlapA72.yAlarm
AND  %cn8.cc1.2
ST   %PLCerr21.22

LD   ForceFlapUpZone
ST   ForceFlapUp_72

********************************************************************************
* Ax73, Unloader Flap L3
********************************************************************************
LD   %ax73.ra4
GT  (
     LD  UnloadSupQta
     ADD 1000
)
OR   Fun_M993_Ch0
ST   ForceFlapUpZone

LD   FlapL3JogHome
OR   AllFlapsHome
OR   ForceFlapUpZone
OR   ParkAllCmd
ST   FlapA73.xManualPlus

LD   FlapL3JogIncline
OR   AllFlapsIncline
ANDN ForceFlapUpZone
ST   FlapA73.xManualMinus

LD   Fun_M987_Ch0                     ** Auto Up command for supports
OR   ForceFlapUpZone
OR   AllFlapsHome
ST   FlapA73.xAutoPlus

LD   Fun_M988_Ch0                     ** Auto DWN command for supports
OR   InclineFlapL3_ISO
ANDN ForceFlapUpZone
ST   FlapA73.xAutoMinus

LD   I_I_FlapL3_Home
ST   FlapA73.xSensorPlus

LD   I_I_FlapL3_Inclined                ** M57.1
ST   FlapA73.xSensorMinus

CAL  FlapA73

LD   FlapA73.yPistonPlus
OR   HoldFlapInclined
ST   O_O_FlapL3_Home

LD   FlapA73.yPistonMinus
ANDN HoldFlapInclined
ST   O_O_FlapL3_Incline

LD   FlapA73.yAlarm
AND  %cn8.cc1.3
ST   %PLCerr21.26

LD   ForceFlapUpZone
ST   ForceFlapUp_73

********************************************************************************
* Ax74, Unloader Flap L4
********************************************************************************
LD   %ax74.ra4
GT  (
     LD  UnloadSupQta
     ADD 1000
)
OR   Fun_M993_Ch0
ST   ForceFlapUpZone

LD   FlapL4JogHome
OR   AllFlapsHome
OR   ForceFlapUpZone
OR   ParkAllCmd
ST   FlapA74.xManualPlus

LD   FlapL4JogIncline
OR   AllFlapsIncline
ANDN ForceFlapUpZone
ST   FlapA74.xManualMinus

LD   Fun_M989_Ch0                     ** Auto Up command for supports
OR   ForceFlapUpZone
OR   AllFlapsHome
ST   FlapA74.xAutoPlus

LD   Fun_M990_Ch0                     ** Auto DWN command for supports
OR   InclineFlapL4_ISO
ANDN ForceFlapUpZone
ST   FlapA74.xAutoMinus

LD   I_I_FlapL4_Home
ST   FlapA74.xSensorPlus

LD   I_I_FlapL4_Inclined                ** M57.1
ST   FlapA74.xSensorMinus

CAL  FlapA74

LD   FlapA74.yPistonPlus
OR   HoldFlapInclined
ST   O_O_FlapL4_Home

LD   FlapA74.yPistonMinus
ANDN HoldFlapInclined
ST   O_O_FlapL4_Incline

LD   FlapA74.yAlarm
AND  %cn8.cc1.4
ST   %PLCerr21.27

LD   ForceFlapUpZone
ST   ForceFlapUp_74

********************************************************************************
* Ax75, Unloader Flap L5
********************************************************************************
LD   %ax75.ra4
GT  (
     LD  UnloadSupQta
     ADD 1000
)
OR   Fun_M993_Ch0
ST   ForceFlapUpZone

LD   FlapL5JogHome
OR   AllFlapsHome
OR   ForceFlapUpZone
OR   ParkAllCmd
ST   FlapA75.xManualPlus

LD   FlapL5JogIncline
OR   AllFlapsIncline
ANDN ForceFlapUpZone
ST   FlapA75.xManualMinus

LD   Fun_M991_Ch0                     ** Auto Up command for supports
OR   ForceFlapUpZone
OR   AllFlapsHome
ST   FlapA75.xAutoPlus

LD   Fun_M992_Ch0                     ** Auto DWN command for supports
OR   InclineFlapL5_ISO
ANDN ForceFlapUpZone
ST   FlapA75.xAutoMinus

LD   I_I_FlapL5_Home
ST   FlapA75.xSensorPlus

LD   I_I_FlapL5_Inclined                ** M57.1
ST   FlapA75.xSensorMinus

CAL  FlapA75

LD   FlapA75.yPistonPlus
OR   HoldFlapInclined
ST   O_O_FlapL5_Home

LD   FlapA75.yPistonMinus
ANDN HoldFlapInclined
ST   O_O_FlapL5_Incline

LD   FlapA75.yAlarm
AND  %cn8.cc1.5
ST   %PLCerr21.28

LD   ForceFlapUpZone
ST   ForceFlapUp_75

END_FUNCTION

(* ---- userlog.plc ---- *)
******************************************************************
* File USERLOG.PLC
* Version: 1.0
******************************************************************

VAR
#include "Cnc.inc"
#include "Iof.inc"

Appoggio:             BOOL;
R_TRIG_1SEC:          R_TRIG;
TP_PROGRAM_ENDPROD:   TP;
TP_PROGRAM_LOAD:      TP;
F_TRIG_ENDPROD: 	  F_TRIG;
R_TRIG_CONTAFOGLI:    R_TRIG;

END_VAR

VAR_IN_OUT
#include "mem.inc"
END_VAR

#include "Iol.inc"

FUNCTION USERLOGGER

****************************************************
* STATI MACCHINA
****************************************************

* Macchina in emergenza generale

LDN  I_EMERGENZA         *(IW0.14) 1= Macchina accesa
ST   %StateMachine0.0    * Macchina in emergenza generale

* Macchina in idle

LD   %cn0.rc0.12         * Selettore modi operativi su AUT (automatic)
ANDN %cn0.rc8.0          * Programma in corso
OR   %cn0.rc0.8          * Selettore modi operativi su REF (taratura)
ANDN %StateMachine0.6    * Macchina in allarme
ANDN %EventMachine0.0    * Caricamento programma
ANDN %EventMachine0.1    * Fine produzione
ST   %StateMachine0.1    * Macchina in idle

* Macchina in manuale

LD   %cn0.rc0.9          * Selettore modi operativi su JOG (manuale)
ANDN %cn0.rc0.12         * Selettore modi operativi su AUT (automatic)
ANDN %StateMachine0.6    * Macchina in allarme
ST   %StateMachine0.2    * Macchina in manuale

* Macchina in semiautomatico

LD   %cn0.rc0.10         * Selettore modi operativi su INC (inc.fissi)
OR   %cn0.rc0.11         * Selettore modi operativi su MDI (semiautom)
ANDN %StateMachine0.6    * Macchina in allarme
ST   %StateMachine0.3    * Macchina in semiautomatico

* Macchina in automatico

LD   %cn0.rc8.0          * Programma in corso
ANDN %StateMachine0.6    * Macchina in allarme
ST   %StateMachine0.4    * Macchina in automatico

* Macchina in hold

LD   %cn0.rc8.1          * Programma interrotto
ANDN %StateMachine0.6    * Macchina in allarme
ST   %StateMachine0.5    * Macchina in hold

LD   %PLCerr0
OR   %PLCerr1
OR   %PLCerr2
OR   %PLCerr3
OR   %PLCerr4
OR   %PLCerr5
OR   %PLCerr6
NE   0
OR   MACC_ALARM          * (gPlc0.10)Macchina in allarme
ST   %StateMachine0.6    * Macchina in allarme

****************************************************
* EVENTI MACCHINA
****************************************************
* Caricamento programma

CAL   TP_PROGRAM_ENDPROD( IN=%ui16.30, PT=2500 ) * Impulso caricamento programma

CAL   F_TRIG_ENDPROD( CLK=TP_PROGRAM_ENDPROD.Q )

CAL   TP_PROGRAM_LOAD( IN=F_TRIG_ENDPROD.Q, PT=2500)

LD    TP_PROGRAM_LOAD.Q
ST    %EventMachine0.0    * Caricamento programma

LD    F_TRIG_ENDPROD.Q
JMPCN AZZERAFOGLI

LD    0
ST    %CounterMachine6

AZZERAFOGLI:

* Fine produzione

LD    TP_PROGRAM_ENDPROD.Q
ST    %EventMachine0.1    * Fine produzione

LD   M30_CN0             * (M0.13) M30:   EndProgram CN0
ANDN ExeAuxMode          * (gPlc0.29)Esecuzione ausiliaria 1000.PGM
ST   Appoggio

CAL R_TRIG_CONTAFOGLI(CLK=Appoggio)

LD  R_TRIG_CONTAFOGLI.Q
JMPCN NOCONTAFOGLI

LD    %CounterMachine6
ADD   1
ST    %CounterMachine6

NOCONTAFOGLI:

*************************************************************************************
* CONTATORI PER DATALOGGER
*************************************************************************************

CAL   R_TRIG_1SEC(CLK=%PLCFLAGS.10)

* Tempo lavoro

LD    R_TRIG_1SEC.Q
AND   %cn0.rc8.0         * Programma in corso
ANDN  %cn0.rc8.1         * Programma interrotto
JMPCN TEMPOLAVORO

LD    %CounterMachine0
ADD   1
ST    %CounterMachine0

TEMPOLAVORO:

* Tempo attrezzaggio

LD    %cn0.rc0.8         * Selettore modi operativi su REF (taratura)
OR    %cn0.rc0.10        * Selettore modi operativi su INC (inc.fissi)
OR    %cn0.rc0.11        * Selettore modi operativi su MDI (semiautom)
AND   R_TRIG_1SEC.Q
JMPCN TEMPOATTREZZAGGIO

LD    %CounterMachine1
ADD   1
ST    %CounterMachine1

TEMPOATTREZZAGGIO:

* Tempo macchina in idle

LD    R_TRIG_1SEC.Q
AND  %StateMachine0.1    * Macchina in idle
JMPCN TEMPOPROGRAMMAZIONE

LD    %CounterMachine2
ADD   1
ST    %CounterMachine2

TEMPOPROGRAMMAZIONE:

* Tempom acchina in allarme

LD    R_TRIG_1SEC.Q
AND  %StateMachine0.6    * Macchina in allarme
JMPCN TEMPOALLARME

LD    %CounterMachine3
ADD   1
ST    %CounterMachine3

TEMPOALLARME:

* Tempo macchina in manuale

LD    R_TRIG_1SEC.Q
AND  %StateMachine0.2    * Macchina in manuale
JMPCN TEMPOFERMA

LD    %CounterMachine4
ADD   1
ST    %CounterMachine4

TEMPOFERMA:

* Tempo macchina in hold

LD    R_TRIG_1SEC.Q
AND  %StateMachine0.5    * Macchina in hold
JMPCN TEMPOHOLD

LD    %CounterMachine5
ADD   1
ST    %CounterMachine5

TEMPOHOLD:

LD    %UserCmdExt.0      * Comando Reset Contatori(se serve lo comanda il server)
JMPCN RESCOUNTER

LD    0
ST    %CounterMachine0
ST    %CounterMachine1
ST    %CounterMachine2
ST    %CounterMachine3
ST    %CounterMachine4
ST    %CounterMachine5

LD    %PLCFLAGS.1
S     %UserCmdInt.0      * Ack Comando Reset Contatori

RESCOUNTER:

LDN   %UserCmdExt.0      * Comando Reset Contatori(se serve lo comanda il server)
R     %UserCmdInt.0     * Ack Comando Reset Contatori

* SEZIONE EVENTI

LD    %PLCerr0
OR    %PLCerr1
OR    %PLCerr2
OR    %PLCerr3
OR    %PLCerr4
OR    %PLCerr5
OR    %PLCerr6
OR    %PLCerr7
OR    %PLCerr20
OR    %PLCerr21
ST    %M104.0          * Riepilogativo allarmi PLC

LD    %PilzSrv.PilzErrCodes0
NE    0
OR(
LD    %PilzSrv.PilzErrCodes1
NE    0
)
OR(
LD    %PilzSrv.PilzErrCodes2
NE    0
)
ST    %M104.1          * Riepilogativo allarmi PLC Safe

LD    %ax0.ra6
NE    0
OR(
LD    %ax1.ra6
NE    0
)
OR(
LD    %ax2.ra6
NE    0
)
OR(
LD    %ax3.ra6
NE    0
)
OR(
LD    %ax4.ra6
NE    0
)
OR(
LD    %ax5.ra6
NE    0
)
OR(
LD    %ax6.ra6
NE    0
)
OR(
LD    %ax7.ra6
NE    0
)
OR(
LD    %ax8.ra6
NE    0
)
OR(
LD    %ax9.ra6
NE    0
)
OR(
LD    %ax10.ra6
NE    0
)
OR(
LD    %ax11.ra6
NE    0
)
OR(
LD    %ax12.ra6
NE    0
)
OR(
LD    %ax13.ra6
NE    0
)
OR(
LD    %ax14.ra6
NE    0
)
OR(
LD    %ax15.ra6
NE    0
)
OR(
LD    %ax16.ra6
NE    0
)
OR(
LD    %ax17.ra6
NE    0
)
OR(
LD    %ax18.ra6
NE    0
)
OR(
LD    %ax19.ra6
NE    0
)
OR(
LD    %ax20.ra6
NE    0
)
OR(
LD    %ax21.ra6
NE    0
)
OR(
LD    %ax22.ra6
NE    0
)
OR(
LD    %ax23.ra6
NE    0
)
OR(
LD    %ax24.ra6
NE    0
)
OR(
LD    %ax25.ra6
NE    0
)
OR(
LD    %ax26.ra6
NE    0
)
OR(
LD    %ax27.ra6
NE    0
)
OR(
LD    %ax28.ra6
NE    0
)
OR(
LD    %ax29.ra6
NE    0
)
OR(
LD    %ax30.ra6
NE    0
)
OR(
LD    %ax31.ra6
NE    0
)
OR(
LD    %ax32.ra6
NE    0
)
OR(
LD    %ax33.ra6
NE    0
)
OR(
LD    %ax34.ra6
NE    0
)
OR(
LD    %ax35.ra6
NE    0
)
OR(
LD    %ax36.ra6
NE    0
)
OR(
LD    %ax37.ra6
NE    0
)
OR(
LD    %ax38.ra6
NE    0
)
OR(
LD    %ax39.ra6
NE    0
)
OR(
LD    %ax40.ra6
NE    0
)
OR(
LD    %ax41.ra6
NE    0
)
OR(
LD    %ax54.ra6
NE    0
)
OR(
LD    %ax72.ra6
NE    0
)
ST    %M104.2          * Riepilogativo allarmi assi

LD    %cn0.rc8.3
OR    %cn1.rc8.3
OR    %cn2.rc8.3
OR    %cn3.rc8.3
OR    %cn4.rc8.3
OR    %cn5.rc8.3
OR    %cn7.rc8.3
OR    %cn8.rc8.3
ST    %M104.3          * Riepilogativo allarmi canale

* FINE SEZIONE EVENTI

END_FUNCTION

(* ---- usrCh6.plc ---- *)
*******************************************************************************
*******************************************************************************
*   @@@ CH6: LOG and COM Function Requests
*******************************************************************************
*******************************************************************************
#funcdec "assi.plc"
#funcdec "cnc.plc"
#funcdec "DynMng.plc"
#funcdec "FBAux.plc"
#funcdec "SupForce.plc"

#include "usrMem.inc"
#include "iol.inc"

VAR_IN_OUT
#include "mem.inc"
#include "usrIol.inc"
END_VAR

VAR
#include "cnc.inc"

Ax60PosEnd:         BOOL;
Ax61PosEnd:         BOOL;

TON_CH6_RUN_STP:    TON;        * TON for CH6_RUN_STP
RTRIG_CH6_RUN_STP:  R_TRIG;     * RTRIG for CH6_RUN_STP
FTRIG_CH6_RUN_STP:  F_TRIG;     * FTRIG for CH6_RUN_STP

GESTCH6:            GESTCH;
CH6END:             GESTCHEND;
GESTAX60:           GESTAX;
GESTAX61:           GESTAX;
PRS_AX60:           AX_PRESET;
PRS_AX61:           AX_PRESET;
CYCOMSUP:           CALC_CYCOMSUP;
CYCOMSUP_UN:        CALC_CYCOMSUP;
END_VAR

FUNCTION CH6

PATH %cn6

LD   ON_ONE_SCAN                   ** PLCFLAGS.8  Flag on alla prima scansione PLC
R    UI_CH6_RUN_STP                ** (M1.0) START/STOP channel 6

CAL  TON_CH6_RUN_STP(IN=ALWAYS_ONE,PT=3000) ** TON for CH6_RUN_STP
CAL  RTRIG_CH6_RUN_STP(CLK:=TON_CH6_RUN_STP.Q) ** RTRIG for CH6_RUN_STP
CAL  FTRIG_CH6_RUN_STP(CLK:=UI_CH6_RUN_STP) ** FTRIG for CH6_RUN_STP

LD   RTRIG_CH6_RUN_STP.Q
OR   UI_CH6_RUN_STP                ** (M1.0) START/STOP channel 6
S    CH6_RUN_STP                   ** (M1.1) START/STOP channel 6 flag

LD   FTRIG_CH6_RUN_STP.Q
OR   ON_ONE_SCAN                   ** PLCFLAGS.8  Flag on alla prima scansione PLC
R    CH6_RUN_STP                   ** (M1.1) START/STOP channel 6 flag

LD   ALWAYS_ONE                    ** PLCFLAGS.1  Flag sempre stato on
ST   GESTCH6.xCmdFromInput        * Disabilita comandi standard macchina
ST   GESTCH6.xSelFromInput        * Disabilita selezioni standard macchina

LD   %PLCFLAGS.0                  ** Condizioni richiesta hold canale 0
ST   GESTCH6.xHold                * comando Hold al canale (esterno)
ST   GESTCH6.xEmer                * comando Emergenza al canale (esterno)
ST   GESTCH6.xBlkSearch
ST   GESTCH6.xIntBlkSrc           * Forzam. esec. ricerca blocco interna

LD   ALWAYS_ONE                    ** PLCFLAGS.1  Flag sempre stato on
ST   GESTCH6.xSelAUT             * selezione modo AUT (con sel. esterna)

LDN  CH6_RUN_STP                   ** (M1.1) START/STOP channel 6 flag
ST   GESTCH6.xReset               * comando RESET al canale (esterno)

LD   CH6_RUN_STP                   ** (M1.1) START/STOP channel 6 flag
ST   GESTCH6.xStart

LD   ChannelFeedrate               ** feedrate for channel
ST   GESTCH6.xOverride            * override assi (esterno)

LD   CH6_RUN_STP                   ** (M1.1) START/STOP channel 6 flag
JMPC InRun

LD   -1
ST   GESTCH6.xPPNumber            * numero part program da eseguire
JMP  ComRS

InRun:
LD   6666
ST   GESTCH6.xPPNumber            * numero part program da eseguire

ComRS:

LD   ALWAYS_ONE                   ** PLCFLAGS.1  Flag sempre stato on
ST   GESTCH6.xCmdFromInput

CAL  GESTCH6

LDN  BCO_PRGRUN			          ** rc8.0  Programma in corso
AND  TON_CH6_RUN_STP.Q
ST   %PLCerr0.16                  ** canale 6 in STOP

*******************************************************************************
*   Virtual X axis for motor cylinder composite support quota (Loader)
*******************************************************************************
PATH %ax60

LD   %cc1.0                        * Maschera assi associata al canale 0
JMPCN NOAX60

LD   ALWAYS_ONE                    ** PLCFLAGS.1  Flag sempre stato on
ST   GESTAX60.xZeroForced          * Forzamento asse tarato
ST   GESTAX60.xLockRef             * Blocco avvio ciclo REF da canale
ST   GESTAX60.xEnFIR               * Abilita filtri FIR
ST   GESTAX60.xEnFrComp            ** Abilita friction compensation
ST   GESTAX60.xDisLimiter

LD   Res_Axes                      ** (gPlc25.1) reset axes disable electric shaft
ST   GESTAX60.xUnlock

* LD   %rc8.3                        * Current channel in alarm
* OR   %cn0.rc8.3                    * ch0 in alarm
* OR   %cn3.rc8.3                    * ch3 in alarm
* ST   GESTAX60.xSetAlarm            ** Forzamento allarme asse

*   Virtual X Quota Preset

LDN  Ax60PosEnd
ANDN Pul_Reset
ST   PRS_AX60.xax_ENABLE
ST   GESTAX60.xFromPlc

LDN  PRS_AX60.xax_ENABLE
OR   Pul_Reset
ST   PRS_AX60.xax_CLEAR

LD   PRS_AX60.xax_ENABLE
AND  PRS_AX60.yax_READY
ANDN PRS_AX60.yax_ENDERR
ST   PRS_AX60.xax_START

*LD   %pa9
*ST   PRS_AX60.xax_VEL

CAL  CYCOMSUP(xLenCy:=CyComLenLoader, xEnCyTubeSiz:=EnCyComTubeDim, xAxNum:=60)

LD   CYCOMSUP.yModeCode.1
JMPCN _OFTLOADER
     LD   CyComLenLoader
	 MUL  1000
     ST   PRS_AX60.xax_QUOTA
_OFTLOADER:

LD   CYCOMSUP.yModeCode.0
ORN  %config_machine0.7
JMPCN _NO_OFTLOADER
     LD   0
     ST   PRS_AX60.xax_QUOTA
_NO_OFTLOADER:

LD   CYCOMSUP.yModeCode.2
AND  %config_machine0.7
ST   %PLCerr20.27

LD   %ra24
SUB  PRS_AX60.xax_QUOTA
ABS
LT   100
ST   Ax60PosEnd

CAL  GESTAX60
CAL  PRS_AX60

NOAX60:

*******************************************************************************
*   Virtual Y axis for motor cylinder composite support quota (Unloader)
*******************************************************************************
PATH %ax61

LD   %cc1.1                        * Maschera assi associata al canale 0
JMPCN NOAX61

LD   ALWAYS_ONE                    ** PLCFLAGS.1  Flag sempre stato on
ST   GESTAX61.xZeroForced          * Forzamento asse tarato
ST   GESTAX61.xLockRef             * Blocco avvio ciclo REF da canale
ST   GESTAX61.xEnFIR               * Abilita filtri FIR
ST   GESTAX61.xEnFrComp            ** Abilita friction compensation
ST   GESTAX61.xDisLimiter

LD   Res_Axes                      ** (gPlc25.1) reset axes disable electric shaft
ST   GESTAX61.xUnlock

* LD   %rc8.3                        * Current channel in alarm
* OR   %cn0.rc8.3                    * ch0 in alarm
* OR   %cn3.rc8.3                    * ch3 in alarm
* ST   GESTAX61.xSetAlarm            ** Forzamento allarme asse

*   Virtual Y Quota Preset

LDN  Ax61PosEnd
ANDN Pul_Reset
ST   PRS_AX61.xax_ENABLE
ST   GESTAX61.xFromPlc

LDN  PRS_AX61.xax_ENABLE
OR   Pul_Reset
ST   PRS_AX61.xax_CLEAR

LD   PRS_AX61.xax_ENABLE
AND  PRS_AX61.yax_READY
ANDN PRS_AX61.yax_ENDERR
ST   PRS_AX61.xax_START

*LD   %pa9
*ST   PRS_AX61.xax_VEL

CAL  CYCOMSUP_UN(xLenCy:=CyComLenUnloader, xEnCyTubeSiz:=EnCyComTubeDimUn, xAxNum:=61)

LD   CYCOMSUP_UN.yModeCode.1
JMPCN _OFTUNLOADER
     LD   CyComLenUnloader
	 MUL  1000
     ST   PRS_AX61.xax_QUOTA
_OFTUNLOADER:

LD   CYCOMSUP_UN.yModeCode.0
ORN  %config_machine0.8
JMPCN _NO_OFTUNLOADER
     LD   0
     ST   PRS_AX61.xax_QUOTA
_NO_OFTUNLOADER:

LD   CYCOMSUP_UN.yModeCode.2
AND  %config_machine0.8
ST   %PLCerr20.28

LD   %ra24
SUB  PRS_AX61.xax_QUOTA
ABS
LT   100
ST   Ax61PosEnd

CAL  GESTAX61
CAL  PRS_AX61

NOAX61:

**************************
* Acknowledg funzioni "M"
**************************
*
LD   %PLCFLAGS.0
ST   CH6END.xWaitMFun

CAL  CH6END

END_FUNCTION

(* ---- usrCh7.plc ---- *)
*******************************************************************************
*******************************************************************************
*   @@@ CH7: Horizontal Unloading Supports
*******************************************************************************
*******************************************************************************
#funcdec "assi.plc"
#funcdec "cnc.plc"

#include "iol.inc"
#include "usrMem.inc"

VAR_IN_OUT
#include "mem.inc"
#include "usrIol.inc"

ActualQtaAbsRef     AT %pa18;                       * Absolute homing quota
QtaRefAbsSet        AT %LsPlc50;                    * Absolute homing quota setting
END_VAR

VAR
#include "cnc.inc"

GESTCH7:            GESTCH;
CH7END:             GESTCHEND;
GESTAX85:           GESTAX;
GESTAX86:           GESTAX;
GESTAX87:           GESTAX;
GESTAX88:           GESTAX;

AXLSREF85:          AX_LS_REF;
AXLSREF86:          AX_LS_REF;
AXLSREF87:          AX_LS_REF;
AXLSREF88:          AX_LS_REF;

RTRIG_AX_SEL85:     R_TRIG;
RTRIG_AX_SEL86:     R_TRIG;
RTRIG_AX_SEL87:     R_TRIG;
RTRIG_AX_SEL88:     R_TRIG;

UnSupp_85_GoUp:     BOOL;
UnSupp_86_GoUp:     BOOL;
UnSupp_87_GoUp:     BOOL;
UnSupp_88_GoUp:     BOOL;

END_VAR

FUNCTION CH7

PATH %cn7

LD   ALWAYS_ONE                                     ** PLCFLAGS.1  Flag sempre stato on
ST   GESTCH7.xCmdFromInput

LD   ALWAYS_ONE                                     ** PLCFLAGS.1  Flag sempre stato on
ST   GESTCH7.xEscOpCmd

LD   %PLCFLAGS.0
ST   GESTCH7.xSelFromInput                          * Disabilita selezioni standard macchina

LD   Ch0_Ref_Gen
ST   GESTCH7.xSelREF

LD   Ch0_Ref_Sin
ST   GESTCH7.xSingleRef

LD   Ch0_Jog
ST   GESTCH7.xSelJOG

LD   Ch0_Inc
ST   GESTCH7.xSelINC

LD   Ch0_Auto
ST   GESTCH7.xSelAUT

LD   ProgRunCh0
ANDN %cn0.rc8.1
ANDN PlcEmerGen                                     ** M0.10 Emergenza generale
OR (
LD   Start_Ch0
AND  ch7_in_ref
)
OR(
LD   Start_Ch0
AND  BCI_MDI                                        ** rc0.11  Selettore modi operativi su MDI (semiautom)
AND (
 LD  UP_SELCHAN                                     ** ui17 Canale selezionato da monitor canale
 EQ  7
)
)
ST   GESTCH7.xStart                                 * comando START al canale (esterno)

LD   ResetChannels
ST   GESTCH7.xReset                                 * comando RESET al canale (esterno)

LD   %cn0.rc8.1                                    ** Condizioni richiesta hold canale 0
OR(
LD   Pul_Stop_Req
AND  BCI_MDI                                        ** rc0.11  Selettore modi operativi su MDI (semiautom)
)
ST   GESTCH7.xHold                                  * comando Hold al canale (esterno)

LD   Ch0Alarm
ST   GESTCH7.xEmer                                  * comando Emergenza al canale (esterno)

LD   7777
ST   GESTCH7.xPPNumber                              * numero part program da eseguire

LD   %PLCFLAGS.0
ST   GESTCH7.xBlkSearch
ST   GESTCH7.xIntBlkSrc                             * Forzam. esec. ricerca blocco interna
ST   GESTCH7.xOverstore                             * Ab. overstore dopo ricerca blocco (provv.)

LD   MainChFeedrate                                 ** feedrate for channel
ST   GESTCH7.xOverride

CAL  GESTCH7

LD   GESTCH7.yProgramRun                            * Programma in corso
ST   PRGRUN_CN8

LD   BCO_STB_GET                                    ** rc8.17 Strobe per GET resources
AND  AxStopSincGRPMacc                              ** (gPlc13.11)Assi Fermi per sincronismo GRP[ax]
ST   BCI_ACK_GET                                    ** rc0.29  ACK per GET resource

********************************************************************************
* Unload Horizontal Axes
********************************************************************************
PATH %ax85
PATH %ax_lsref85

***************************************
*   POWER ON (PON)
***************************************
LD   %pa3.31                                        * Simulato
ORN  %cc1.2                                         * Maschera assi associata al canale
OR(
LD   %nvel11                                        ** 3,4=CANopen, Ecat
EQ   3
)
OR(
LD   %nvel11                                        ** 3,4=CANopen, Ecat
EQ   4
)
ST   Pon_UnSupp_85                                  ** PON unload support axis
***************************************

LD  %cc1.2                                          * Maschera assi associata al canale 8
JMPCN NOAX85

***
*   LIMIT SWITCH & REFERENCE SWITCH

LD   %lsrefmode
ST   AXLSREF85.x_REF_mode                           * 0=use ref switch...

LD   %lsreflevel
ST   AXLSREF85.x_TYPE_LS                            * (1=NC, 0=NO)

LD   I_I_AX85_NEG
ST   AXLSREF85.x_MIN_LS                             * Min Limit switch

LD   I_I_AX85_POS                * C saw minimumm limit switchV
ST   AXLSREF85.x_MAX_LS                             * Max Limit switch

LD   ALWAYS_ZERO
ST   AXLSREF85.x_REF_S                              * Reference switch

CAL  AXLSREF85

LD   AXLSREF85.y_MIN_LS                             * Min Limit switch
ST   GESTAX85.xMinusLS                              * Negative limit switch

LD   AXLSREF85.y_MAX_LS                             * Max Limit switch
ST   GESTAX85.xPlusLS                               * Positive limit switch

LD   AXLSREF85.y_REF_S                              * Reference switch
ST   GESTAX85.xRefLS                                * Reference
***

LD   MainAxesPowerAllowed
AND  MainAxesPower                                  * PON
ST   GESTAX85.xCloseLoop

LD   Sel_Z_Ch7
ST   GESTAX85.xSelected

***************************************
* Change REF quota for ABS reference
***************************************
CAL  RTRIG_AX_SEL85(CLK:=GESTAX85.xSelected)

LD   RTRIG_AX_SEL85.Q
JMPCN NoSel85
LD   ActualQtaAbsRef                                ** Absolute homing quota
ST   QtaRefAbsSet                                   ** Absolute homing quota setting
NoSel85:

LD   GESTAX85.xSelected
AND  %nvel14.0                                      * Se Vale 1 ?gestito "Encoder Assoluto" (Da Configura Asse)
AND (
LD   ActualQtaAbsRef                                ** Absolute homing quota
NE   QtaRefAbsSet                                   ** Absolute homing quota setting
)
JMPCN NoEq85

LD   QtaRefAbsSet                                   ** Absolute homing quota setting
ST   ActualQtaAbsRef                                ** Absolute homing quota
NoEq85:
***************************************

LD   Pul_Jogp                                       ** (gPlc0.4)jog+ pushbutton
AND  GESTAX85.xSelected
ANDN PlcEmerGen                                     ** M0.10 Emergenza generale
AND  GESTAX85.xCloseLoop
ST   GESTAX85.xJogPlus

LD   Pul_Jogm                                       ** (gPlc0.5)jog- pushbutton
AND  GESTAX85.xSelected
ANDN PlcEmerGen                                     ** M0.10 Emergenza generale
AND  GESTAX85.xCloseLoop
ST   GESTAX85.xJogMinus

LD   %nvel14.0                                      * Se Vale 1 ?gestito "Encoder Assoluto" (Da Configura Asse)
ST   GESTAX85.xZeroForced                           * Forzamento asse tarato

LD   GESTAX2_xHoldMoving                            * Richiesta blocco avanzamento
OR   HoldSuppUn_HorAx85
ST   GESTAX85.xHoldMoving                           * Richiesta blocco avanzamento

LD   Res_Axes                                       ** (gPlc25.1) reset axes disable electric shaft
ST   GESTAX85.xUnlock

LDN  ch8_in_ref                                     ** channel 3 in ref
ST   GESTAX85.xEnFIR                                * Abilita filtri FIR
ST   GESTAX85.xEnFrComp                             ** Abilita friction compensation

LD   ALWAYS_ZERO                                    ** PLCFLAGS.0  Flag sempre stato off
ST   GESTAX85.xDisLimiter

LD   %cn0.rc8.3                                     * ch0 in alarm
OR   %cn3.rc8.3                                     * ch3 in alarm
ST   GESTAX85.xSetAlarm                             ** Forzamento allarme asse

LD   usrReqGrantSupHorAx85
ST   GESTAX85.xFromPlc

CAL  GESTAX85

LD   GESTAX85.yDriveNotEn
S    %PLCerr3.16                                     * Axis 85, drive not enable

LD   TON_ABIL_PON
ANDN Pon_UnSupp_85
ST   %PLCerr3.20

LD   BSG_INC                                        ** rg1.2 Selezione modo INC (inc.fissi)
JMPCN SVIX85

LD   %pa59                                          * Velocit?di Repos
MUL  1000
DIV  60
MUL  MainChFeedrate                                 ** (gPlc16) feed degli assi (%)
DIV  100
ST   %ra50                                          * Limitazione velocita' massima interpolazione

SVIX85:
NOAX85:

********************************************************************************
* Unload Support 1 (ax86)
********************************************************************************
PATH %ax86
PATH %ax_lsref86

***************************************
*   POWER ON (PON)
***************************************
LD   %pa3.31            * Simulato
ORN  %cc1.3             * Maschera assi associata al canale
OR(
LD   %nvel11            ** 3,4=CANopen, Ecat
EQ   3
)
OR(
LD   %nvel11            ** 3,4=CANopen, Ecat
EQ   4
)
ST   Pon_UnSupp_86      ** PON unload support axis
***************************************

LD   %cc1.3           * Maschera assi associata al canale 8
JMPCN NOAX86

***
*   LIMIT SWITCH & REFERENCE SWITCH

LD   %lsrefmode
ST   AXLSREF86.x_REF_mode        * 0=use ref switch...

LD   %lsreflevel
ST   AXLSREF86.x_TYPE_LS         * (1=NC, 0=NO)

LD   I_I_AX86_NEG
ST   AXLSREF86.x_MIN_LS          * Min Limit switch

LD   I_I_AX86_POS
ST   AXLSREF86.x_MAX_LS          * Max Limit switch

LD   ALWAYS_ZERO
ST   AXLSREF86.x_REF_S           * Reference switch

CAL  AXLSREF86

LD   AXLSREF86.y_MIN_LS          * Min Limit switch
ST   GESTAX86.xMinusLS           * Negative limit switch

LD   AXLSREF86.y_MAX_LS          * Max Limit switch
ST   GESTAX86.xPlusLS            * Positive limit switch

LD   AXLSREF86.y_REF_S           * Reference switch
ST   GESTAX86.xRefLS             * Reference
***

LD   MainAxesPowerAllowed
AND  MainAxesPower               * PON
ST   GESTAX86.xCloseLoop

LD   Sel_U_Ch7
ST   GESTAX86.xSelected

***************************************
* Change REF quota for ABS reference
***************************************
CAL  RTRIG_AX_SEL86(CLK:=GESTAX86.xSelected)

LD   RTRIG_AX_SEL86.Q
JMPCN NoSel86
LD   ActualQtaAbsRef               ** Absolute homing quota
ST   QtaRefAbsSet                  ** Absolute homing quota setting
NoSel86:

LD   GESTAX86.xSelected
AND  %nvel14.0                     * Se Vale 1 � gestito "Encoder Assoluto" (Da Configura Asse)
AND (
LD   ActualQtaAbsRef               ** Absolute homing quota
NE   QtaRefAbsSet                  ** Absolute homing quota setting
)
JMPCN NoEq86

LD   QtaRefAbsSet                  ** Absolute homing quota setting
ST   ActualQtaAbsRef               ** Absolute homing quota
NoEq86:
***************************************

LD   Pul_Jogp                      ** (gPlc0.4)jog+ pushbutton
AND  GESTAX86.xSelected
ANDN PlcEmerGen                      ** M0.10 Emergenza generale
AND  GESTAX86.xCloseLoop
ST   GESTAX86.xJogPlus

LD   Pul_Jogm                      ** (gPlc0.5)jog- pushbutton
AND  GESTAX86.xSelected
ANDN PlcEmerGen                      ** M0.10 Emergenza generale
AND  GESTAX86.xCloseLoop
ST   GESTAX86.xJogMinus

LD   %nvel14.0                     * Se Vale 1 � gestito "Encoder Assoluto" (Da Configura Asse)
ST   GESTAX86.xZeroForced          * Forzamento asse tarato

LD   GESTAX2_xHoldMoving           * Richiesta blocco avanzamento
OR   HoldSuppUn_HorAx86
ST   GESTAX86.xHoldMoving          * Richiesta blocco avanzamento

LD   Res_Axes                      ** (gPlc25.1) reset axes disable electric shaft
ST   GESTAX86.xUnlock

LDN  ch8_in_ref                    ** channel 3 in ref
ST   GESTAX86.xEnFIR               * Abilita filtri FIR
ST   GESTAX86.xEnFrComp            ** Abilita friction compensation

LD   ALWAYS_ZERO                   ** PLCFLAGS.0  Flag sempre stato off
ST   GESTAX86.xDisLimiter

LD   %cn0.rc8.3                    * ch0 in alarm
OR   %cn3.rc8.3                    * ch3 in alarm
**OR   EmerINC
ST   GESTAX86.xSetAlarm            ** Forzamento allarme asse

LD   usrReqGrantSupHorAx86
ST   GESTAX86.xFromPlc

CAL  GESTAX86

LD   GESTAX86.yDriveNotEn
S    %PLCerr3.17                    * Axis 86, drive not enable

LD   TON_ABIL_PON
ANDN Pon_UnSupp_86
ST   %PLCerr3.21

LD   BSG_INC                       ** rg1.2 Selezione modo INC (inc.fissi)
JMPCN SVIX86

LD   %pa59                         * Velocit� di Repos
MUL  1000
DIV  60
MUL  MainChFeedrate                ** (gPlc16) feed degli assi (%)
DIV  100
ST   %ra50                         * Limitazione velocita' massima interpolazione

SVIX86:
NOAX86:

********************************************************************************
* Unload Support 2 (ax87)
********************************************************************************
PATH %ax87
PATH %ax_lsref87

***************************************
*   POWER ON (PON)
***************************************
LD   %pa3.31                                        * Simulato
ORN  %cc1.4                                         * Maschera assi associata al canale
OR(
LD   %nvel11                                        ** 3,4=CANopen, Ecat
EQ   3
)
OR(
LD   %nvel11                                        ** 3,4=CANopen, Ecat
EQ   4
)
ST   Pon_UnSupp_87                                  ** PON unload support axis
***************************************

LD  %cc1.4                                          * Maschera assi associata al canale 8
JMPCN NOAX87

***
*   LIMIT SWITCH & REFERENCE SWITCH

LD   %lsrefmode
ST   AXLSREF87.x_REF_mode                           * 0=use ref switch...

LD   %lsreflevel
ST   AXLSREF87.x_TYPE_LS                            * (1=NC, 0=NO)

LD   I_I_AX87_NEG
ST   AXLSREF87.x_MIN_LS                             * Min Limit switch

LD   I_I_AX87_POS                                  * W maximun limit switch
ST   AXLSREF87.x_MAX_LS                             * Max Limit switch

LD   ALWAYS_ZERO
ST   AXLSREF87.x_REF_S                              * Reference switch

CAL  AXLSREF87

LD   AXLSREF87.y_MIN_LS                             * Min Limit switch
ST   GESTAX87.xMinusLS                              * Negative limit switch

LD   AXLSREF87.y_MAX_LS                             * Max Limit switch
ST   GESTAX87.xPlusLS                               * Positive limit switch

LD   AXLSREF87.y_REF_S                              * Reference switch
ST   GESTAX87.xRefLS                                * Reference
***

LD   MainAxesPowerAllowed
AND  MainAxesPower                                  * PON
ST   GESTAX87.xCloseLoop

LD   Sel_V_Ch7
ST   GESTAX87.xSelected

***************************************
* Change REF quota for ABS reference
***************************************
CAL  RTRIG_AX_SEL87(CLK:=GESTAX87.xSelected)

LD   RTRIG_AX_SEL87.Q
JMPCN NoSel87
LD   ActualQtaAbsRef                                ** Absolute homing quota
ST   QtaRefAbsSet                                   ** Absolute homing quota setting
NoSel87:

LD   GESTAX87.xSelected
AND  %nvel14.0                                      * Se Vale 1 ?gestito "Encoder Assoluto" (Da Configura Asse)
AND (
LD   ActualQtaAbsRef                                ** Absolute homing quota
NE   QtaRefAbsSet                                   ** Absolute homing quota setting
)
JMPCN NoEq87

LD   QtaRefAbsSet                                   ** Absolute homing quota setting
ST   ActualQtaAbsRef                                ** Absolute homing quota
NoEq87:
***************************************

LD   Pul_Jogp                                       ** (gPlc0.4)jog+ pushbutton
AND  GESTAX87.xSelected
ANDN PlcEmerGen                                     ** M0.10 Emergenza generale
AND  GESTAX87.xCloseLoop
ST   GESTAX87.xJogPlus

LD   Pul_Jogm                                       ** (gPlc0.5)jog- pushbutton
AND  GESTAX87.xSelected
ANDN PlcEmerGen                                     ** M0.10 Emergenza generale
AND  GESTAX87.xCloseLoop
ST   GESTAX87.xJogMinus

LD   %nvel14.0                                      * Se Vale 1 ?gestito "Encoder Assoluto" (Da Configura Asse)
ST   GESTAX87.xZeroForced                           * Forzamento asse tarato

LD   GESTAX2_xHoldMoving                            * Richiesta blocco avanzamento
OR   HoldSuppUn_HorAx87
ST   GESTAX87.xHoldMoving                           * Richiesta blocco avanzamento

LD   Res_Axes                                       ** (gPlc25.1) reset axes disable electric shaft
ST   GESTAX87.xUnlock

LDN  ch8_in_ref                                     ** channel 3 in ref
ST   GESTAX87.xEnFIR                                * Abilita filtri FIR
ST   GESTAX87.xEnFrComp                             ** Abilita friction compensation

LD   ALWAYS_ZERO                                    ** PLCFLAGS.0  Flag sempre stato off
ST   GESTAX87.xDisLimiter

LD   %cn0.rc8.3                                     * ch0 in alarm
OR   %cn3.rc8.3                                     * ch3 in alarm
ST   GESTAX87.xSetAlarm                             ** Forzamento allarme asse

LD   usrReqGrantSupHorAx87
ST   GESTAX87.xFromPlc

CAL  GESTAX87

LD   GESTAX87.yDriveNotEn
S    %PLCerr3.18                                     * Axis 87, drive not enable

LD   TON_ABIL_PON
ANDN Pon_UnSupp_87
ST   %PLCerr3.22

LD   BSG_INC                                        ** rg1.2 Selezione modo INC (inc.fissi)
JMPCN SVIX87

LD   %pa59                                          * Velocit?di Repos
MUL  1000
DIV  60
MUL  MainChFeedrate                                 ** (gPlc16) feed degli assi (%)
DIV  100
ST   %ra50                                          * Limitazione velocita' massima interpolazione

SVIX87:
NOAX87:

********************************************************************************
* Unload Support 3 (ax88)
********************************************************************************
PATH %ax88
PATH %ax_lsref88

***************************************
*   POWER ON (PON)
***************************************
LD   %pa3.31                                        * Simulato
ORN  %cc1.4                                         * Maschera assi associata al canale
OR(
LD   %nvel11                                        ** 3,4=CANopen, Ecat
EQ   3
)
OR(
LD   %nvel11                                        ** 3,4=CANopen, Ecat
EQ   4
)
ST   Pon_UnSupp_88                                  ** PON unload support axis
***************************************

LD  %cc1.5                                          * Maschera assi associata al canale 8
JMPCN NOAX88

***
*   LIMIT SWITCH & REFERENCE SWITCH

LD   %lsrefmode
ST   AXLSREF88.x_REF_mode                           * 0=use ref switch...

LD   %lsreflevel
ST   AXLSREF88.x_TYPE_LS                            * (1=NC, 0=NO)

LD   I_I_AX88_NEG
ST   AXLSREF88.x_MIN_LS                             * Min Limit switch

LD   I_I_AX88_POS
ST   AXLSREF88.x_MAX_LS                             * Max Limit switch

LD   ALWAYS_ZERO
ST   AXLSREF88.x_REF_S                              * Reference switch

CAL  AXLSREF88

LD   AXLSREF88.y_MIN_LS                             * Min Limit switch
ST   GESTAX88.xMinusLS                              * Negative limit switch

LD   AXLSREF88.y_MAX_LS                             * Max Limit switch
ST   GESTAX88.xPlusLS                               * Positive limit switch

LD   AXLSREF88.y_REF_S                              * Reference switch
ST   GESTAX88.xRefLS                                * Reference
***

LD   MainAxesPowerAllowed
AND  MainAxesPower                                  * PON
ST   GESTAX88.xCloseLoop

LD   Sel_W_Ch7
ST   GESTAX88.xSelected

***************************************
* Change REF quota for ABS reference
***************************************
CAL  RTRIG_AX_SEL88(CLK:=GESTAX88.xSelected)

LD   RTRIG_AX_SEL88.Q
JMPCN NoSel88
LD   ActualQtaAbsRef                                ** Absolute homing quota
ST   QtaRefAbsSet                                   ** Absolute homing quota setting
NoSel88:

LD   GESTAX88.xSelected
AND  %nvel14.0                                      * Se Vale 1 ?gestito "Encoder Assoluto" (Da Configura Asse)
AND (
LD   ActualQtaAbsRef                                ** Absolute homing quota
NE   QtaRefAbsSet                                   ** Absolute homing quota setting
)
JMPCN NoEq88

LD   QtaRefAbsSet                                   ** Absolute homing quota setting
ST   ActualQtaAbsRef                                ** Absolute homing quota
NoEq88:
***************************************

LD   Pul_Jogp                                       ** (gPlc0.4)jog+ pushbutton
AND  GESTAX88.xSelected
ANDN PlcEmerGen                                     ** M0.10 Emergenza generale
AND  GESTAX88.xCloseLoop
ST   GESTAX88.xJogPlus

LD   Pul_Jogm                                       ** (gPlc0.5)jog- pushbutton
AND  GESTAX88.xSelected
ANDN PlcEmerGen                                     ** M0.10 Emergenza generale
AND  GESTAX88.xCloseLoop
*ANDN CMD_HOLDMOVING_CH8.4
ST   GESTAX88.xJogMinus

LD   %nvel14.0                                      * Se Vale 1 ?gestito "Encoder Assoluto" (Da Configura Asse)
ST   GESTAX88.xZeroForced                           * Forzamento asse tarato

LD   GESTAX2_xHoldMoving                            * Richiesta blocco avanzamento
OR   HoldSuppUn_HorAx88
ST   GESTAX88.xHoldMoving                           * Richiesta blocco avanzamento

LD   Res_Axes                                       ** (gPlc25.1) reset axes disable electric shaft
ST   GESTAX88.xUnlock

LDN  ch8_in_ref                                     ** channel 3 in ref
ST   GESTAX88.xEnFIR                                * Abilita filtri FIR
ST   GESTAX88.xEnFrComp                             ** Abilita friction compensation

LD   ALWAYS_ZERO                                    ** PLCFLAGS.0  Flag sempre stato off
ST   GESTAX88.xDisLimiter

LD   %cn0.rc8.3                                     * ch0 in alarm
OR   %cn3.rc8.3                                     * ch3 in alarm
**OR   EmerINC
ST   GESTAX88.xSetAlarm                             ** Forzamento allarme asse

LD   usrReqGrantSupHorAx88
ST   GESTAX88.xFromPlc

CAL  GESTAX88

LD   GESTAX88.yDriveNotEn
S    %PLCerr3.19                                     * Axis 88, drive not enable

LD   TON_ABIL_PON
ANDN Pon_UnSupp_88
ST   %PLCerr3.23

LD   BSG_INC                                        ** rg1.2 Selezione modo INC (inc.fissi)
JMPCN SVIX88

LD   %pa59                                          * Velocit?di Repos
MUL  1000
DIV  60
MUL  MainChFeedrate                                 ** (gPlc16) feed degli assi (%)
DIV  100
ST   %ra50                                          * Limitazione velocita' massima interpolazione

SVIX88:
NOAX88:

**************************
* Acknowledg funzioni "M"
**************************
*
LD   %PLCFLAGS.0
ST   CH7END.xWaitMFun

CAL  CH7END

END_FUNCTION
